// Mitsubishi GX Works2 project: DryChaomer   PLC: FX3G

TYPE stSTEP : STRUCT
  iRiseTime : INT;
  iHoldTime : INT;
  iHoldTempr : INT;
  iHoldHumid : INT;
  iEnable : INT;
  iVFDSpeed : INT;
END_STRUCT END_TYPE

TYPE stSTEPHelper : STRUCT
  iState : INT;  (* 0 - Idle, 1 - Raise, 2 - Hold, 3 - Done *)
END_STRUCT END_TYPE

// global labels: GVL
VAR_GLOBAL
  gxReset AT M400 : BOOL;
  gxStart AT M401 : BOOL;
END_VAR
VAR_GLOBAL CONSTANT
  c_STATE_IDLE : INT;
  c_STATE_RAISE : INT := 1;
  c_STATE_HOLD : INT := 2;
  c_STATE_DONE : INT := 3;
  c_STEP_NUM : INT := 4;
END_VAR
VAR_GLOBAL
  grSteps : ARRAY [0..4] OF stSTEP;
  giCS_Num AT D1000 : INT;  (* Текущий номер этапа *)
  giCS_RaiseETime AT D1001 : INT;  (* Время подъема текущего этапа прошедшее *)
  giCS_HoldETime AT D1002 : INT;  (* Время удержания текущего этапа прошедшее *)
  giPID_T_SV : INT;  (* ПИД температура уставка *)
  giPID_T_PV : INT;  (* ПИД температура текущее значение *)
  giPID_T_MV : INT;  (* ПИД температура задача на выход *)
  giPID_H_SV : INT;  (* ПИД влажность уставка *)
  giPID_H_PV : INT;  (* ПИД влажность текущее значение *)
  giPID_H_MV : INT;  (* ПИД влажность задача на выход *)
  giStart_T : INT;  (* Значение с которого нужно начинать подъем температуры на этапе подъема *)
  giStart_H : INT;  (* Значение с которого нужно начинать подъем влажности на этапе подъема *)
  griTLimit AT R31 : INT;  (* Delta for limit for PID *)
  griHLimit AT R32 : INT;  (* Delta for limit for PID *)
  gxPIDANTemp AT M402 : BOOL;  (* Включить автонастройку для ПИД температуры *)
  gxPIDANHum AT M403 : BOOL;  (* Включить автонастройку для ПИД влажности *)
  gxPIDANModeTemp AT M404 : BOOL;  (* 0 - limit cycle, 1 - step response *)
  gxPIDANModeHum AT M405 : BOOL;  (* 0 - limit cycle, 1 - step response *)
  garstStepHelper : ARRAY [0..4] OF stSTEPHelper;
  gxDone AT M406 : BOOL;  (* Закончили процесс сушки *)
  giProbeType : INT;  (* 0 - avrage, 1-2 tempr *)
  gxVFD1 AT M420 : BOOL;
  gxVFD2 AT M421 : BOOL;
  gxVFD3 AT M422 : BOOL;
  gxVFD4 AT M423 : BOOL;
  gxVFD5 AT M424 : BOOL;
  gxVFD6 AT M425 : BOOL;
  gxVFD7 AT M426 : BOOL;
  gxVFD8 AT M427 : BOOL;
  gxVFD9 AT M428 : BOOL;
  gxVFD10 AT M429 : BOOL;
  gxVFD11 AT M430 : BOOL;
  gxVFD12 AT M431 : BOOL;
  gxVFD13 AT M432 : BOOL;
  gxVFD14 AT M433 : BOOL;
  giCSVFDSpeed AT D1003 : INT;  (* Скорость ПЧ текущего этапа *)
  griMinVentSpeed AT R33 : INT;  (* Minimum speed of humid vent in % *)
  griMinVentDelay AT R34 : INT;  (* Minimum time to delay before turn on after PID is 0 *)
  gxAlarmReset AT M434 : BOOL;
  giCSTemp_SV AT D1004 : INT;  (* Уставка температуры текущего этапа *)
  giCSHum_SV AT D1005 : INT;  (* Уставка влажности текущего этапа *)
  giCSRaiseTime AT D1001 : INT;  (* Время подъема текущего этапа *)
  giCSHoldTime AT D1002 : INT;  (* Время удержания текущего этапа *)
  giRaiseET : INT;  (* Осталось времени подъема в процентах 0-100 *)
  giHoldET : INT;  (* Осталось времени удержания в процентах 0-100 *)
  giPID_T_P AT R503 : INT;  (* ПИД Пропроциональный *)
  giPID_T_I AT R504 : INT;  (* ПИД Интегральный *)
  giPID_T_D AT R506 : INT;  (* ПИД Диференциальный *)
  giPID_H_P AT R603 : INT;  (* ПИД Пропроциональный *)
  giPID_H_I AT R604 : INT;  (* ПИД Интегральный *)
  giPID_H_D AT R606 : INT;  (* ПИД Диференциальный *)
  gxProgress AT M435 : BOOL;  (* В процессе находимся *)
END_VAR

// global labels: IO
VAR_GLOBAL
  AO_Valve1 AT D8052 : INT;
  AO_Valve2 AT D8053 : INT;
  AO_VFD1 AT R23750 : INT;
  AO_VFD2 AT R23751 : INT;
  AO_VFD3 AT R23752 : INT;
  AO_VFD4 AT R23753 : INT;
  AO_VFD5 AT R23754 : INT;
  AO_VFD6 AT R23755 : INT;
  AO_VFD7 AT R23756 : INT;
  AO_VFD8 AT R23757 : INT;
  AO_VFD9 AT R23758 : INT;
  AO_VFD10 AT R23759 : INT;
  AO_VFD11 AT R23760 : INT;
  AO_VFD12 AT R23761 : INT;
  AO_VFD13 AT R23762 : INT;
  AO_VFD14 AT R23763 : INT;
  AO_VFDVent AT R23764 : INT;
  AI_Temp1 AT D0 : INT;  (* Тепература 1 в контуре 1 *)
  AI_Temp2 AT D1 : INT;  (* Тепература 2 в контуре 1 *)
  AI_Temp3 AT D2 : INT;  (* Тепература 1 в контуре 2 *)
  AI_Temp4 AT D3 : INT;  (* Тепература 2 в контуре 2 *)
  AI_TempProd1 AT D4 : INT;  (* Температура продукта 1 *)
  AI_TempProd2 AT D5 : INT;  (* Температура продукта 2 *)
  AI_TempProd3 AT D6 : INT;  (* Температура продукта 3 *)
  DI_OverheatCP AT X000 : BOOL;  (* Перегрев ШУ *)
  DI_RKF AT X001 : BOOL;
  DI_OverheatPU AT X002 : BOOL;  (* Перегрев СШ *)
  DI_VFDAlarm1 AT X003 : BOOL;
  DI_VFDAlarm2 AT X004 : BOOL;
  DI_VFDAlarm3 AT X005 : BOOL;
  DI_VFDAlarm4 AT X006 : BOOL;
  DI_VFDAlarm5 AT X007 : BOOL;
  DI_VFDAlarm6 AT X010 : BOOL;
  DI_VFDAlarm7 AT X011 : BOOL;
  DI_VFDAlarm8 AT X012 : BOOL;
  DI_VFDAlarm9 AT X020 : BOOL;
  DI_VFDAlarm10 AT X021 : BOOL;
  DI_VFDAlarm11 AT X022 : BOOL;
  DI_VFDAlarm12 AT X023 : BOOL;
  DI_VFDAlarm13 AT X024 : BOOL;
  DI_VFDAlarm14 AT X025 : BOOL;
  DI_VFDAlarmHumid AT X026 : BOOL;
  DI_Door AT X030 : BOOL;
  DO_VFD1 AT Y000 : BOOL;
  DO_VFD2 AT Y001 : BOOL;
  DO_VFD3 AT Y002 : BOOL;
  DO_VFD4 AT Y003 : BOOL;
  DO_VFD5 AT Y004 : BOOL;
  DO_VFD6 AT Y005 : BOOL;
  DO_VFD7 AT Y006 : BOOL;
  DO_VFD8 AT Y007 : BOOL;
  DO_VFD9 AT Y010 : BOOL;
  DO_VFD10 AT Y011 : BOOL;
  DO_VFD11 AT Y012 : BOOL;
  DO_VFD12 AT Y013 : BOOL;
  DO_VFD13 AT Y020 : BOOL;
  DO_VFD14 AT Y021 : BOOL;
  DO_VFDHum AT Y022 : BOOL;
  DO_Red AT Y023 : BOOL;
  DO_Green AT Y024 : BOOL;
  DO_Yellow AT Y025 : BOOL;
  DO_Buzzer AT Y026 : BOOL;
  DO_VFDReset AT Y030 : BOOL;
  AI_Pressure AT D9 : INT;  (* Давление *)
  AI_AirFlow AT D10 : INT;  (* Проток *)
  AI_Valve1Position AT D11 : INT;  (* Положения клапана задвижки *)
  AI_Valve2Position AT D12 : INT;  (* Положение клапана задвижки *)
  AI_PVTTempr AT D7 : INT;  (* Температура *)
  AI_PVTHumid AT D8 : INT;  (* Влажность *)
END_VAR

// task Task_01 (event TRUE, interval 0, priority 31): POU_01
// task INIT (event M8002, interval 0, priority 29): INIT
// task PROCES (event FALSE, interval T#50ms, priority 31): PROCESS
// task TCO (event I650, interval 0, priority 21): TCO_TICKER_50
// user libraries (not included): AlarmManger128v14, Modbusv16, TimeControl50, Utils

PROGRAM POU_01
VAR
  iStep : INT;
  fbAmBlock : AM_IS_BLOCK;
  iCount : INT;
  iLastStep : INT;
  xPIDTEnable : BOOL;
  xPIDHEnable : BOOL;
  fbTPVentDelay : TP;
END_VAR
fbAmBlock(iProcessNum:=0,iSeverity:=0);
MOV(fbAmBlock.Q AND iStep > 2, 40, iStep);

xPIDTEnable := iStep = 20 OR iStep = 30 AND (giPID_T_PV < (giPID_T_SV + griTLimit));
xPIDHEnable := iStep = 20 OR iStep = 30  AND NOT fbTPVentDelay.Q AND (giPID_H_PV > (giPID_H_SV - griHLimit));
fbTPVentDelay(IN := MEF(DO_VFDHum), PT:= MIN_TO_TIME(griMinVentDelay));
PID(xPIDTEnable, giPID_T_SV, giPID_T_PV, R500, giPID_T_MV);
PID(xPIDHEnable, giPID_H_SV, giPID_H_PV, R600, giPID_H_MV);
MOV(NOT xPIDTEnable, 0, giPID_T_MV);
MOV(NOT xPIDHEnable, 0, giPID_H_MV);

CASE iStep OF
	0: (* Init *)
		iStep := 1;

	1: (* Reset *)
		giStart_T := 0;
		giStart_H := 0;
		gxDone := FALSE;
		gxProgress := FALSE;
		FOR iCount := 0 TO 4 DO
			garstStepHelper[iCount].iState := c_STATE_IDLE;
		END_FOR;
		iStep := 2;

	2: (* Idle *)
		IF gxStart AND NOT fbAmBlock.Q THEN
			iLastStep := 4;
			FOR iCount := 0 TO 4 DO
				IF grSteps[4 - iCount].iEnable = 1 THEN
					iLastStep := 4 - iCount;
					EXIT;
				END_IF;
			END_FOR;
			IF gxPIDANTemp THEN
	            R501 := 2#0000_0000_0011_0001; (* Autotune Step Response *)
	            IF NOT gxPIDANModeTemp THEN
	                R501 := 2#0000_0000_0111_0001; (* Autotune limit cycle *)
	            END_IF;
	            gxPIDANTemp := FALSE;
	        END_IF;
	        IF gxPIDANHum THEN
	            R601 := 2#0000_0000_0011_0000; (* Autotune Step Response *)
	            IF NOT gxPIDANModeHum THEN
	                R601 := 2#0000_0000_0111_0000; (* Autotune limit cycle *)
	            END_IF;
	            gxPIDANHum := FALSE;
	        END_IF;
			iStep := 10;
			gxProgress := TRUE;
		END_IF;
		
	10: (* Step select *)
	
		FOR iCount := 0 TO 4 DO
			IF grSteps[iCount].iEnable = 1 AND garstStepHelper[iCount].iState < c_STATE_DONE THEN
				
				(* по умолчанию на подъем начала этапа или востановление подъема, 
				но если мы вернулись например после перезагрузки на этап удержания на удержание. *)
				iStep := 20;
				MOV(garstStepHelper[iCount].iState = c_STATE_HOLD, 30, iStep);
				
				IF iStep > 10 THEN
					giCS_Num := iCount;			
					MOV(iStep = 20, c_STATE_RAISE, garstStepHelper[iCount].iState);
					MOV(iStep = 30, c_STATE_HOLD, garstStepHelper[iCount].iState);
					MOV(giStart_T = 0, giPID_T_PV, giStart_T);
					MOV(giStart_H = 0, giPID_H_PV, giStart_H);
					(* Сбрасываем счечтики только если мы начинаем шаг заново. 
					Если мы в него возвращаемся нжно сохранить счет. *)
					IF garstStepHelper[iCount].iState = c_STATE_IDLE THEN
						giCS_RaiseETime := 0;
						giCS_HoldETime := 0;
					END_IF;
					giCSRaiseTime := grSteps[iCount].iRiseTime;
					giCSHoldTime := grSteps[iCount].iHoldTime;
					giCSTemp_SV := grSteps[iCount].iHoldTempr;
					giCSHum_SV := grSteps[iCount].iHoldHumid;
					giCSVFDSpeed := grSteps[iCount].iVFDSpeed;
					EXIT;
				END_IF;
			END_IF;
		END_FOR;
		MOV(iStep = 10, 50, iStep);
		
	
	20: (* Raise *)
		INCP(M8014, giCS_RaiseETime);

		giPID_T_SV := SCALE(giCS_RaiseETime, 0, grSteps[giCS_Num].iRiseTime, giStart_T, grSteps[giCS_Num].iHoldTempr);
		giPID_H_SV := SCALE(giCS_RaiseETime, 0, grSteps[giCS_Num].iRiseTime, giStart_H, grSteps[giCS_Num].iHoldHumid);

		giRaiseET := WORK_LEFT(grSteps[giCS_Num].iRiseTime, giCS_RaiseETime);
		MOV(giCS_RaiseETime >= grSteps[giCS_Num].iRiseTime, 30, iStep);
		MOV(iStep = 30, c_STATE_HOLD, garstStepHelper[giCS_Num].iState);
		
	
	30: (* Hold *)
		INCP(M8014, giCS_HoldETime);
		
		giPID_T_SV := grSteps[giCS_Num].iHoldTempr;
		giPID_H_SV := grSteps[giCS_Num].iHoldHumid;
		
		giHoldET := WORK_LEFT(grSteps[giCS_Num].iHoldTime, giCS_HoldETime);
		MOV(giCS_HoldETime >= grSteps[giCS_Num].iHoldTime, 10, iStep);
		MOV(iStep = 10, c_STATE_DONE, garstStepHelper[giCS_Num].iState);
		MOV(iStep = 10, grSteps[giCS_Num].iHoldTempr, giStart_T);
		MOV(iStep = 10, grSteps[giCS_Num].iHoldHumid, giStart_H);

	40: (* Pause *)
		MOV(NOT fbAmBlock.Q, 10, iStep);

	50: (* Finish *)
		gxDone := TRUE;
		MOV(NOT gxStart, 1, iStep);
	
END_CASE;
END_PROGRAM

PROGRAM INIT
VAR
  fbAmInit : AM_INIT;
END_VAR
AM_D_START := 3000;

(* Init PID *) (* Настройка параметров ПИД регулирования *)
R500 := 1000; (* Time 1c *)
R501 := 2#0000_0000_0000_0001; (* Heating mode *)
R522 := 4000; (* Output max 100% *)
R523 := 0; (* Output min *)
R525 := 10; (* Delta for Autotune 1.0 C *)
R526 := R522; (* Autotune output upper value *)
R527 := 0; (* Autotune output lower value *)

(* Init PIDHum *) (* Настройка параметров ПИД регулирования *)
R600 := 1000; (* Time 1c *)
R601 := 2#0000_0000_0000_0000; (* Cooling mode *)
R622 := 32000; (* Output max 100% *)
R623 := 0; (* Output min *)
R625 := 10; (* Delta for Autotune 1.0 C *)
R626 := R622; (* Autotune output upper value *)
R627 := 0; (* Autotune output lower value *)



fbAmInit.iProcess  := 0;
fbAmInit.iSeverity := 0;

fbAmInit(iNum:=0,xLatch:=0,xBuzzer:=0,xLock:=0);
fbAmInit(iNum:=1,xLatch:=0,xBuzzer:=0,xLock:=0);
fbAmInit(iNum:=2,xLatch:=0,xBuzzer:=0,xLock:=0);
fbAmInit(iNum:=3,xLatch:=0,xBuzzer:=0,xLock:=0);
fbAmInit(iNum:=4,xLatch:=0,xBuzzer:=0,xLock:=0);
fbAmInit(iNum:=5,xLatch:=0,xBuzzer:=0,xLock:=0);
fbAmInit(iNum:=6,xLatch:=0,xBuzzer:=0,xLock:=0);
fbAmInit(iNum:=7,xLatch:=0,xBuzzer:=0,xLock:=0);
fbAmInit(iNum:=8,xLatch:=0,xBuzzer:=0,xLock:=0);
fbAmInit(iNum:=9,xLatch:=0,xBuzzer:=0,xLock:=0);
fbAmInit(iNum:=10,xLatch:=0,xBuzzer:=0,xLock:=0);
fbAmInit(iNum:=11,xLatch:=0,xBuzzer:=0,xLock:=0);
fbAmInit(iNum:=12,xLatch:=0,xBuzzer:=0,xLock:=0);
fbAmInit(iNum:=13,xLatch:=0,xBuzzer:=0,xLock:=0);
fbAmInit(iNum:=14,xLatch:=0,xBuzzer:=0,xLock:=0);
END_PROGRAM

PROGRAM PROCESS
VAR
  fbAmSet : AM_SET;
  fbAmReset : AM_RST;
  fbTPVentDelay : TP;
END_VAR
CASE giProbeType OF
	0: giPID_T_PV := (AI_Temp1 + AI_Temp2) / 2;
	1: giPID_T_PV := AI_Temp1;
	2: giPID_T_PV := AI_Temp2;
END_CASE;

AI_Temp1 := R23700;
AI_Temp2 := R23701;
AI_Temp3 := R23702;
AI_Temp4 := R23703;
AI_TempProd1 := R23704;
AI_TempProd2 := R23705;
AI_TempProd3 := R23706;
AI_Pressure := SCALE(R23708, 0, 32000, 0, -1000);
AI_PVTHumid := SCALE(R23709, 0, 32000, 0, 100);
AI_PVTTempr := SCALE(R23710, 0, 32000, -500,1200);
AI_AirFlow  := SCALE(R23711, 0, 32000, 0, 100);

D6032 := D8032;
D6033 := D8033;
AI_Valve1Position := SCALE(D8032,0,4000,0,100);
AI_Valve2Position := SCALE(D8033,0,4000,0,100);

D6034 := D8052;
D6035 := D8053;
giPID_H_PV := AI_PVTHumid;
AO_Valve1 := giPID_T_MV;
AO_Valve2 := giPID_T_MV;

fbAmReset(IN:= gxAlarmReset);

fbAmSet(iNum:=0,xState:=DI_VFDAlarm1);
fbAmSet(iNum:=1,xState:=DI_VFDAlarm2);
fbAmSet(iNum:=2,xState:=DI_VFDAlarm3);
fbAmSet(iNum:=3,xState:=DI_VFDAlarm4);
fbAmSet(iNum:=4,xState:=DI_VFDAlarm5);
fbAmSet(iNum:=5,xState:=DI_VFDAlarm6);
fbAmSet(iNum:=6,xState:=DI_VFDAlarm7);
fbAmSet(iNum:=7,xState:=DI_VFDAlarm8);
fbAmSet(iNum:=8,xState:=DI_VFDAlarm9);
fbAmSet(iNum:=9,xState:=DI_VFDAlarm10);
fbAmSet(iNum:=10,xState:=DI_VFDAlarm11);
fbAmSet(iNum:=11,xState:=DI_VFDAlarm12);
fbAmSet(iNum:=12,xState:=DI_VFDAlarm13);
fbAmSet(iNum:=13,xState:=DI_VFDAlarm14);
fbAmSet(iNum:=14,xState:=DI_VFDAlarmHumid);

BMOV(TRUE, D3280, 8, K4M2000);

AO_VFD1 := SCALE(giCSVFDSpeed,0,100,0,32000);
DO_VFD1 := gxVFD1 AND NOT DI_VFDAlarm1 AND (AO_VFD1 > 0);

AO_VFD2 := SCALE(giCSVFDSpeed,0,100,0,32000);
DO_VFD2 := gxVFD2 AND NOT DI_VFDAlarm2 AND (AO_VFD2 > 0);

AO_VFD3 := SCALE(giCSVFDSpeed,0,100,0,32000);
DO_VFD3 := gxVFD3 AND NOT DI_VFDAlarm3 AND (AO_VFD3 > 0);

AO_VFD4 := SCALE(giCSVFDSpeed,0,100,0,32000);
DO_VFD4 := gxVFD4 AND NOT DI_VFDAlarm4 AND (AO_VFD4 > 0);

AO_VFD5 := SCALE(giCSVFDSpeed,0,100,0,32000);
DO_VFD5 := gxVFD5 AND NOT DI_VFDAlarm5 AND (AO_VFD5 > 0);

AO_VFD6 := SCALE(giCSVFDSpeed,0,100,0,32000);
DO_VFD6 := gxVFD6 AND NOT DI_VFDAlarm6 AND (AO_VFD6 > 0);

AO_VFD7 := SCALE(giCSVFDSpeed,0,100,0,32000);
DO_VFD7 := gxVFD7 AND NOT DI_VFDAlarm7 AND (AO_VFD7 > 0);

AO_VFD8 := SCALE(giCSVFDSpeed,0,100,0,32000);
DO_VFD8 := gxVFD8 AND NOT DI_VFDAlarm8 AND (AO_VFD8 > 0);

AO_VFD9 := SCALE(giCSVFDSpeed,0,100,0,32000);
DO_VFD9 := gxVFD9 AND NOT DI_VFDAlarm9 AND (AO_VFD9 > 0);

AO_VFD10 := SCALE(giCSVFDSpeed,0,100,0,32000);
DO_VFD10 := gxVFD10 AND NOT DI_VFDAlarm10 AND (AO_VFD10 > 0);

AO_VFD11 := SCALE(giCSVFDSpeed,0,100,0,32000);
DO_VFD11 := gxVFD11 AND NOT DI_VFDAlarm11 AND (AO_VFD11 > 0);

AO_VFD12 := SCALE(giCSVFDSpeed,0,100,0,32000);
DO_VFD12 := gxVFD12 AND NOT DI_VFDAlarm12 AND (AO_VFD12 > 0);

AO_VFD13 := SCALE(giCSVFDSpeed,0,100,0,32000);
DO_VFD13 := gxVFD13 AND NOT DI_VFDAlarm13 AND (AO_VFD13 > 0);

AO_VFD14 := SCALE(giCSVFDSpeed,0,100,0,32000);
DO_VFD14 := gxVFD14 AND NOT DI_VFDAlarm14 AND (AO_VFD14 > 0);


AO_VFDVent := giPID_H_MV;
(* Если нужно ограничивать, и есть значение приводим его к минимальному. *)
LIMITATION_E(griMinVentSpeed > 0 AND giPID_H_MV > 0, SCALE(griMinVentSpeed,0,100,0,32000), giPID_H_MV, 32000, AO_VFDVent);
DO_VFDHum := NOT DI_VFDAlarmHumid AND AO_VFDVent > 0;
END_PROGRAM
